// TIA Portal V20 export
DATA_BLOCK "Settings"   // DB6
{ DB_Accessible_From_OPC_UA := 'FALSE' }
// stored: DBAccessibleFromOPCUA false, DBAccessibleFromWebserver false, MemoryReserve 100
   VAR
      diagPlc : "LAF_typePlcDiag";   // HMI Schnittstelle PLC Diagnose / HMI interface PLC diag
      checksum : "LAF_typeChecksum";   // HMI Schnittstelle PLCChecksum / HMI interface PLCChecksum
      diagMemCard : "LAF_typeMemCardDiag";   // HMI Schnittstelle SMCDiag / HMI interface SMCDiag
      cycleTimes : "LSicar_typeGlobalRuntime";
      setLocalPlcTime : "LAF_typeSetPlcTime";
      ITConnection : Bool := FALSE;   // Provides a visual representation of the connection with the IT systems.
   END_VAR
BEGIN
   diagPlc.manualReadAll := FALSE;
   diagPlc.blockBusyAfterRestart := FALSE;
   diagPlc.im0Data.Manufacturer_ID := 42;
   diagPlc.im0Data.Order_ID := '6ES7 518-3UT10-0AB0 ';
   diagPlc.im0Data.Serial_Number := 'S C-T4A0RVHM2025';
   diagPlc.im0Data.Hardware_Revision := 1;
   diagPlc.im0Data.Software_Revision."Type" := 'V';
   diagPlc.im0Data.Software_Revision.Functional := 4;
   diagPlc.im0Data.Software_Revision.Bugfix := 0;
   diagPlc.im0Data.Software_Revision.Internal := 0;
   diagPlc.im0Data.Revision_Counter := 0;
   diagPlc.im0Data.Profile_ID := 0;
   diagPlc.im0Data.Profile_Specific_Type := 0;
   diagPlc.im0Data.IM_Version := 16#0101;
   diagPlc.im0Data.IM_Supported := 16#000E;
   diagPlc.im1PlantDesignLocIdent := '                                                      ';
   diagPlc.im1PlantDesignation := '                                ';
   diagPlc.im1LocIdent := '                      ';
   diagPlc.im2InstallationDate := '2025-02-24 16:59';
   diagPlc.im3AdditionalInfo := '                                                      ';
   diagPlc.addressMac[0] := 16#30;
   diagPlc.addressMac[1] := 16#B8;
   diagPlc.addressMac[2] := 16#51;
   diagPlc.addressMac[3] := 16#66;
   diagPlc.addressMac[4] := 16#CF;
   diagPlc.addressMac[5] := 16#66;
   diagPlc.addressIpV4[0] := 192;
   diagPlc.addressIpV4[1] := 168;
   diagPlc.addressIpV4[2] := 200;
   diagPlc.addressIpV4[3] := 51;
   diagPlc.addressSubnet[0..2] := 255;
   diagPlc.addressSubnet[3] := 0;
   diagPlc.im0SwRev := 'V';
   checksum.checksumStandard := 'E4AA23DFFDEEA866';
   checksum.checksumStandardOld := 'E4AA23DFFDEEA866';
   checksum.checksumSafety := '0A6CEC4B00000000';
   checksum.checksumSafetyOld := '0A6CEC4B00000000';
   checksum.checksumTextlists := '676DC45055902179';
   checksum.checksumTextlistsOld := '676DC45055902179';
   checksum.dateTimeStandardModified := DT#2026-01-06-00:09:42.545;
   checksum.dateTimeSafetyModified := DT#2026-01-06-00:09:42.545;
   checksum.dateTimeTextlistModified := DT#2026-01-06-00:09:42.545;
   checksum.standardModified := FALSE;
   checksum.safetyModified := FALSE;
   checksum.textlistsModified := FALSE;
   checksum.summaryModified := FALSE;
   checksum.updateValuesOld := FALSE;
   diagMemCard.alarmWarnInfo := 16#00;
   diagMemCard.manualUpdate := FALSE;
   diagMemCard.memorySpaceKbyte := 31151664;
   diagMemCard.assignedMemorySpaceKbyte := 68208;
   diagMemCard.assignedMemorySpace := 0;
   diagMemCard.usedLifetime := 0;
   diagMemCard.paraLifetime := 80;
   diagMemCard.warningFromMemorySpace := 81;
   diagMemCard.alarmFromMemorySpace := 95;
   cycleTimes.prevCycle := 3;
   cycleTimes.reset := FALSE;
   cycleTimes.maxCycle := 5;
   cycleTimes.minCycle := 2;
   cycleTimes.maxCycleRuntime := 100;
   cycleTimes.minCycleRuntime := 1;
   cycleTimes.maxCommRuntime := 0;
   setLocalPlcTime.newDateAndTime := DT#1990-01-01-00:00:00;
   setLocalPlcTime.daylightSavingTime := FALSE;
   setLocalPlcTime.apply := FALSE;
END_DATA_BLOCK
